TYPE ST_ContactDetectOutput :
STRUCT
    (* Force On已经形成尚未确认的Contact候选。 *)
    bCandidate : BOOL;
    (* Contact已经防抖确认。 *)
    bDetected : BOOL;
    (* Contact候选时锁存的压向力，单位kN。 *)
    rCandidateForce_kN : LREAL;
    (* Contact候选时锁存的Z轴绝对位置，单位mm。 *)
    rCandidateAxisPosition_mm : LREAL;
    (* Contact候选时锁存的外部位移绝对位置，单位mm。 *)
    rCandidateSensorPosition_mm : LREAL;
    (* Contact确认时锁存的压向力，单位kN。 *)
    rDetectedForce_kN : LREAL;
    (* Contact确认时锁存的Z轴绝对位置，单位mm。 *)
    rDetectedAxisPosition_mm : LREAL;
    (* Contact确认时锁存的外部位移绝对位置，单位mm。 *)
    rDetectedSensorPosition_mm : LREAL;
    (* Contact确认时仅一个扫描周期的参考点锁存请求。 *)
    bReferenceLatchRequest : BOOL;
    (* 输入无效或检测窗口异常。 *)
    bFault : BOOL;
    (* Contact故障编号，0表示无故障。 *)
    nFaultId : UDINT;
END_STRUCT
END_TYPE

(* stored: Version 1.1.0.1
   DUT ST_ContactDetectOutput: Id {D2000000-0000-4000-8000-000000000010} *)
